# EPICS autosave request: iocBoot/iocoxford/auto_positions.req
file oxford_settings.req P=$(P)
